///Automatically created by BoxConfigurator
VAR_GLOBAL
	///Subsystem number 10 emulation
	fbSubsystem10_Emulation: FB_ProBoxSubsystemEmulation;
END_VAR

(* stored: Version 1.1.0.1, ProductVersion 3.1.4024.9
   GVL SubsystemEmulation: Id {ced514d1-5b5b-4fe7-8242-475e3b40b6f1} *)
